// TIA Portal V19 export
TYPE "LEXCHANGETRAY_typeHandlingXyzEm_toNgConveyorDeliver"
// stored: Access Published
   STRUCT
      feedback : "LEXCHANGETRAY_typeHandlingXyzEm_toNgConveyorFeedback";
      req : "LEXCHANGETRAY_typeHandlingXyzEm_toNgConveyoReq";
   END_STRUCT;
END_TYPE
